(* PLC project Unnamed, Unknown Unnamed 1 *)
(* stored: creationDateTime 2024-10-03T07:24:23, modificationDateTime 2024-10-03T07:24:23 *)

CONFIGURATION Config0
  RESOURCE Res0 ON PLC
  END_RESOURCE
END_CONFIGURATION
